FUNCTION "fcTest" : Void
{ S7_Optimized_Access := 'TRUE' }
VERSION : 0.1
   VAR_INPUT
      in : Bool;
   END_VAR

   VAR_OUTPUT
      out : Bool;
   END_VAR


BEGIN
	#out := #in;
END_FUNCTION

